TYPE "SpeedMachine_CIn"
VERSION : 0.1
// Block: SpeedMachine_CIn
   STRUCT
      Manager : SpeedMachine_CIn_Manager;
      Bwd_ExtEnable : Bool;
      Fwd_ExtEnable : Bool;
      EnableManChangeVel : Bool;
      ExternalPowerOn : Bool;
      ExternalAlarms : Bool;
      VelocityOverride : Struct
         Enable : Bool;
         Value : Real;
      END_STRUCT;
   END_STRUCT;

END_TYPE
